ABB RobotStudio station: Solution_1.rspag

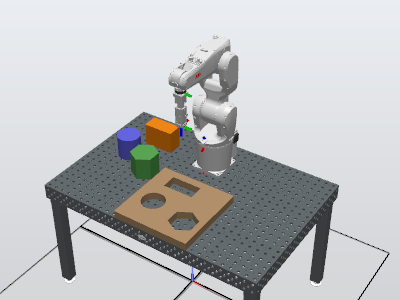
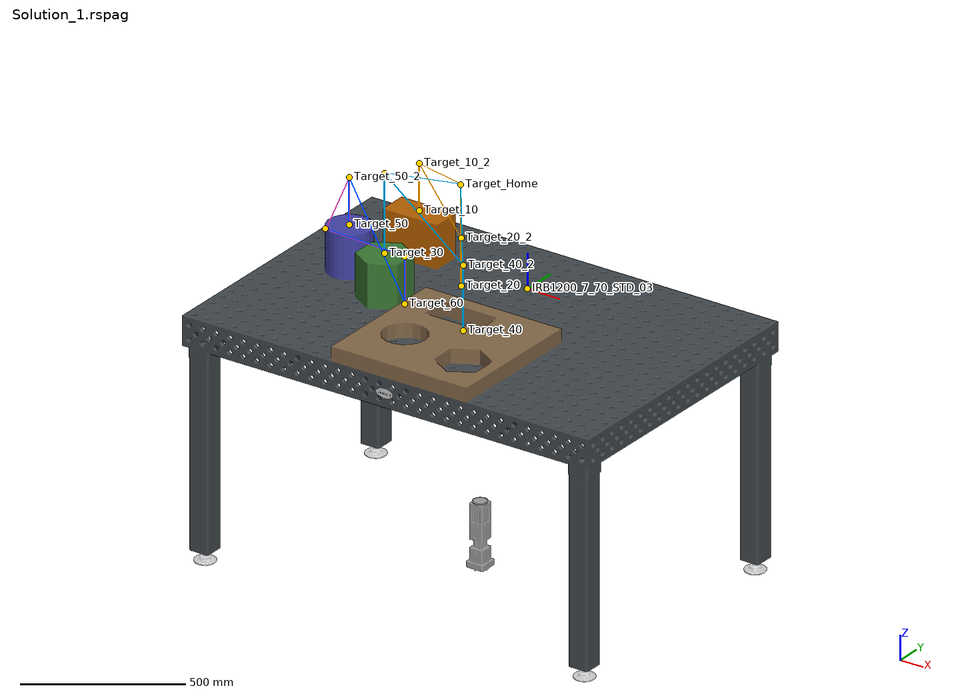
[picture v1: parts stored in the station drawn from their meshes, with robot base, taught points and paths (robot models come from the ABB library and are not in the file)]
--- station ---
Station Solution_1_Tutorial (saved by RobotStudio 22.3.10190.2)
Controller Controller_Solution_1, task T_ROB1: task frame (RAPID world) sits at (0, 250, 830) mm, rotated rx 0 ry 0 rz -90 deg in the station
Controller Controller_Solution_1
  mechanical unit ROB_1: IRB1200_7_70_STD_03, 6 joints, base frame (0, 0, 0) mm
Layout (positions relative to the parent item):
  - table [part] at (-200, -500, 830) mm, size 500 x 500 x 50 mm
  - object_1 [part] at (-600, -150, 830) mm, size 200 x 100 x 150 mm
  - object_2 [part] at (-650, -150, 830) mm, size 149.5 x 149.7 x 150 mm
  - object_3 [part] at (-700, -200, 830) mm, size 155.5 x 179.5 x 150 mm
  - siegmund_1500_1000 [part], size 1500 x 1010.3 x 830 mm
  - object_11 [part] at (-200, -500, 830) mm, size 200 x 100 x 150 mm
  - object_22 [part] at (-200, -500, 830) mm, size 149.5 x 149.7 x 150 mm
  - object_33 [part] at (-200, -500, 830) mm, size 155.5 x 179.5 x 150 mm
  - Assembly2_3 [graphiccomponentgroup] at (-38.87, -9.32, 138.6) mm, rotated rx -90 ry 0 rz 0 deg
    - MHM-32D1-X6400(0):3 [graphiccomponentgroup] at (38.87, 1.1, -15.68) mm, rotated rx 0 ry -90 rz 0 deg
      - _MHM-A3201-1-X6400_DAMPER [part] at (25, -74.2, 0) mm, size 49.7 x 6 x 50 mm
      - _MHM-32D1-X6400(0)_BODY:2 [part] at (25, 0, 25) mm, rotated rx 0 ry 90 rz 0 deg, size 50 x 79.6 x 50 mm
    - M4x10:5 [part] at (39.02, 86.1, -10.68) mm, rotated rx 180 ry 0 rz 0 deg, size 7 x 7 x 14 mm
    - M4x10:7 [part] at (39.02, 36.1, -10.68) mm, rotated rx 180 ry 0 rz 0 deg, size 7 x 7 x 14 mm
    - ITEM30x30x100:3 [part] at (38.87, 106.1, 9.32) mm, rotated rx 0 ry 0 rz -90 deg, size 100 x 30 x 30 mm
    - M5x75:2 [part] at (57.87, 13.1, -9.68) mm, rotated rx -90 ry 0 rz 0 deg, size 8.5 x 8.5 x 25 mm
    - M4x10:8 [part] at (39.02, 86.1, 29.32) mm, size 7 x 7 x 14 mm
    - M4x10:9 [part] at (39.02, 36.1, 29.32) mm, size 7 x 7 x 14 mm
    - M5x75:3 [part] at (19.87, 13.1, 28.32) mm, rotated rx -90 ry 0 rz 0 deg, size 8.5 x 8.5 x 25 mm
    - M5x75:4 [part] at (57.87, 13.1, 28.32) mm, rotated rx -90 ry 0 rz 0 deg, size 8.5 x 8.5 x 25 mm
    - M5x75:5 [part] at (19.87, 13.1, -9.68) mm, rotated rx -90 ry 0 rz 0 deg, size 8.5 x 8.5 x 25 mm
    - KQ2L06-01N:3 [part] at (47.37, -5.7, 30.32) mm, rotated rx 90 ry 0 rz 89.92 deg, size 21.3 x 22.5 x 10.4 mm
    - KQ2L06-01N:4 [part] at (30.37, -64.9, 30.32) mm, rotated rx 90 ry 0 rz 89.92 deg, size 21.3 x 22.5 x 10.4 mm
    - Part_Bottom_Blue:1 [part] at (17.33, 6.1, -15.68) mm, rotated rx 90 ry 0 rz 0 deg, size 50 x 50 x 45 mm
    - Part_Middle_Black:2 [part] at (17.33, 116.1, 34.32) mm, rotated rx -90 ry 0 rz 0 deg, size 50 x 50 x 45 mm
    - Part_Top_Blue:4 [part] at (38.87, 128.6, 9.32) mm, rotated rx 90 ry 0 rz 0 deg, size 63.8 x 63.8 x 17.5 mm
    - M4x25:1 [part] at (19.87, 109.1, -9.68) mm, rotated rx 90 ry 0 rz 0 deg, size 7 x 7 x 29 mm
    - M4x25:2 [part] at (57.87, 109.1, 28.32) mm, rotated rx 90 ry 0 rz 0 deg, size 7 x 7 x 29 mm
    - M4x25:3 [part] at (19.87, 109.1, 28.32) mm, rotated rx 90 ry 0 rz 0 deg, size 7 x 7 x 29 mm
    - M4x25:4 [part] at (57.87, 109.1, -9.68) mm, rotated rx 90 ry 0 rz 0 deg, size 7 x 7 x 29 mm
    - M4_nut:1 [part] at (57.87, 129.7, 28.32) mm, rotated rx 0 ry -14.91 rz 0 deg, size 7 x 2.2 x 8.1 mm
    - M5x16:1 [part] at (50, 128.6, 20.46) mm, rotated rx 90 ry 0 rz 0 deg, size 8.5 x 8.5 x 21 mm
    - M6x16:1 [part] at (63.87, 129.6, 9.32) mm, rotated rx 90 ry 0 rz 0 deg, size 10 x 10 x 22 mm
    - M4_nut:2 [part] at (57.87, 129.7, -9.68) mm, rotated rx 0 ry -14.91 rz 0 deg, size 7 x 2.2 x 8.1 mm
    - M4_nut:3 [part] at (19.87, 129.7, -9.68) mm, rotated rx 0 ry -14.91 rz 0 deg, size 7 x 2.2 x 8.1 mm
    - M4_nut:4 [part] at (19.87, 129.7, 28.32) mm, rotated rx 0 ry -14.91 rz 0 deg, size 7 x 2.2 x 8.1 mm
    - M5x16:2 [part] at (50, 128.6, -1.82) mm, rotated rx 90 ry 0 rz 0 deg, size 8.5 x 8.5 x 21 mm
    - M5x16:3 [part] at (27.73, 128.6, 20.46) mm, rotated rx 90 ry 0 rz 0 deg, size 8.5 x 8.5 x 21 mm
    - M5x16:4 [part] at (27.73, 128.6, -1.82) mm, rotated rx 90 ry 0 rz 0 deg, size 8.5 x 8.5 x 21 mm
    - M6x16:2 [part] at (13.87, 129.6, 9.32) mm, rotated rx 90 ry 0 rz 0 deg, size 10 x 10 x 22 mm
    - M6x16:3 [part] at (38.87, 129.6, -15.68) mm, rotated rx 90 ry 0 rz 0 deg, size 10 x 10 x 22 mm
    - M6x16:4 [part] at (38.87, 129.6, 34.32) mm, rotated rx 90 ry 0 rz 0 deg, size 10 x 10 x 22 mm
  - smc_magnetic_gripper [mechanism] at (0, -101, 1539.1) mm, rotated rx 180 ry 0 rz 90 deg
      TCP smc_magnetic_gripper at (38.87, -79.1, 9.32) mm, rotated rx 90 ry 0 rz 0 deg
      links: Assembly2_3_Merged
  - IRB1200_7_70_STD_03 [mechanism, from %ABB.RobotStudio.Models.IRB1200%\IRB1200_7_70_STD_03.rslib] at (0, 250, 830) mm, rotated rx 0 ry 0 rz -90 deg; joint values [0, 0, 0, 0, 1.5708, 0] (rad or m)
  - Positioner_object_1 [smart component, from Components\Positioner.rslib]
      properties: Object=object_1; Position=[-0.6 -0.15 0.83]; Orientation=[0 0 0]; Reference=Global; ReferenceObject=(none)
  - Attacher_object_1 [smart component, from Components\Attacher.rslib]
      properties: Parent=smc_magnetic_gripper; Flange=0; Child=object_1; Mount=false; Offset=[0 0 0]; Orientation=[0 0 0]
  - Detacher_object_1 [smart component, from Components\Detacher.rslib]
      properties: Child=object_1; KeepPosition=true
  - Positioner_object_2 [smart component, from Components\Positioner.rslib]
      properties: Object=object_2; Position=[-0.65 -0.15 0.83]; Orientation=[0 0 0]; Reference=Global; ReferenceObject=(none)
  - Positioner_object_3 [smart component, from Components\Positioner.rslib]
      properties: Object=object_3; Position=[-0.7 -0.2 0.83]; Orientation=[0 0 0]; Reference=Global; ReferenceObject=(none)
  - Attacher_object_2 [smart component, from Components\Attacher.rslib]
      properties: Parent=smc_magnetic_gripper; Flange=0; Child=object_2; Mount=false; Offset=[0 0 0]; Orientation=[0 0 0]
  - Attacher_object_3 [smart component, from Components\Attacher.rslib]
      properties: Parent=smc_magnetic_gripper; Flange=0; Child=object_3; Mount=false; Offset=[0 0 0]; Orientation=[0 0 0]
  - Detacher_object_2 [smart component, from Components\Detacher.rslib]
      properties: Child=object_2; KeepPosition=true
  - Detacher_object_3 [smart component, from Components\Detacher.rslib]
      properties: Child=object_3; KeepPosition=true
  - Frame_1 [frame] at (0, 0, 217.7) mm
Attachment: smc_magnetic_gripper is attached to IRB1200_7_70_STD_03 / Link6
Station signals: DI reset
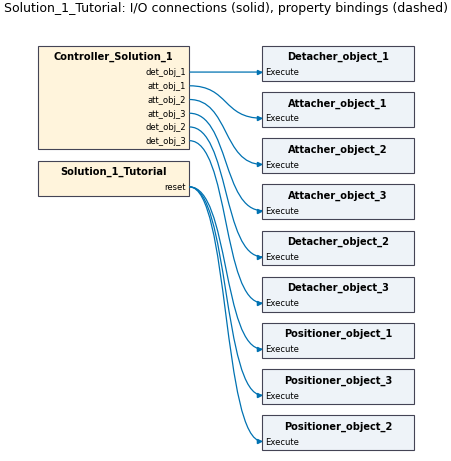
Station logic (signal -> signal, property => property):
  Controller_Solution_1.det_obj_1 -> Detacher_object_1.Execute
  Solution_1_Tutorial.reset -> Positioner_object_1.Execute
  Solution_1_Tutorial.reset -> Positioner_object_3.Execute
  Solution_1_Tutorial.reset -> Positioner_object_2.Execute
  Controller_Solution_1.att_obj_1 -> Attacher_object_1.Execute
  Controller_Solution_1.att_obj_2 -> Attacher_object_2.Execute
  Controller_Solution_1.att_obj_3 -> Attacher_object_3.Execute
  Controller_Solution_1.det_obj_2 -> Detacher_object_2.Execute
  Controller_Solution_1.det_obj_3 -> Detacher_object_3.Execute
Targets, tools, work objects and paths stored in the station and not in the controller backup, written as RAPID:
! task T_ROB1
MODULE CalibData
  PERS tooldata MyTool:=[TRUE,[[31.792631019,0,229.638935148],[0.945518576,0,0.325568154,0]],[1,[0,0,1],[1,0,0,0],0,0,0]];
ENDMODULE


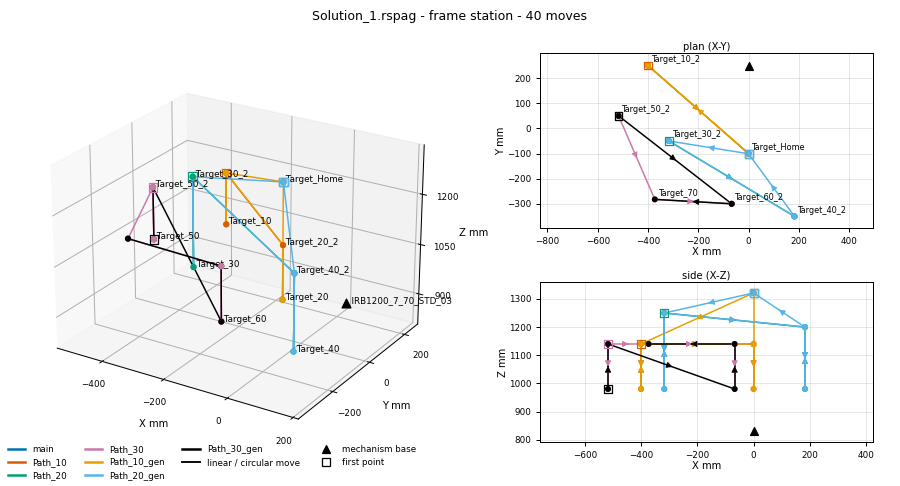
[picture p0: tool path of Solution_1.rspag in frame station, 40 of 40 moves have a stored position in this frame; points joined in program order, loops and branches not executed]
--- Backups/Controller_Solution_1/RAPID/TASK1/PROGMOD/CalibData.modx ---
MODULE CalibData
    PERS tooldata smc_magnetic_gripper:=[TRUE,[[0,0,217.7],[1,0,0,0]],[0.72,[0.001,0.267,107.779],[1,0,0,0],0,0,0]];
ENDMODULE

--- Backups/Controller_Solution_1/RAPID/TASK1/PROGMOD/Module1.modx ---
MODULE Module1
        CONST robtarget Target_Home:=[[351,0,491.4],[0,0,1,0],[-1,0,-1,0],[9E+09,9E+09,9E+09,9E+09,9E+09,9E+09]];
    CONST robtarget Target_10_2:=[[0,-400,310],[0,0,1,0],[-1,0,-2,0],[9E+09,9E+09,9E+09,9E+09,9E+09,9E+09]];
    CONST robtarget Target_10:=[[0,-400,150],[0,0,1,0],[-1,0,-2,0],[9E+09,9E+09,9E+09,9E+09,9E+09,9E+09]];
    CONST robtarget Target_20_2:=[[350,0,310],[0,0,1,0],[0,0,0,0],[9E+09,9E+09,9E+09,9E+09,9E+09,9E+09]];
    CONST robtarget Target_20:=[[350,0,150],[0,0,1,0],[0,0,-1,0],[9E+09,9E+09,9E+09,9E+09,9E+09,9E+09]];
    CONST robtarget Target_30_2:=[[300,-317.298,420],[0,0,1,0],[0,0,0,0],[9E+09,9E+09,9E+09,9E+09,9E+09,9E+09]];
    CONST robtarget Target_30:=[[300,-317.298,150],[0,0,1,0],[0,0,0,0],[9E+09,9E+09,9E+09,9E+09,9E+09,9E+09]];
    CONST robtarget Target_40_2:=[[600,182.702,370],[0,0,1,0],[0,0,0,0],[9E+09,9E+09,9E+09,9E+09,9E+09,9E+09]];
    CONST robtarget Target_40:=[[600,182.702,150],[0,0,1,0],[0,0,0,0],[9E+09,9E+09,9E+09,9E+09,9E+09,9E+09]];
    CONST robtarget Target_50_2:=[[200,-517.298,310],[0,0,1,0],[0,0,0,0],[9E+09,9E+09,9E+09,9E+09,9E+09,9E+09]];
    CONST robtarget Target_60:=[[550,-67.298,150],[0,0,1,0],[0,0,0,0],[9E+09,9E+09,9E+09,9E+09,9E+09,9E+09]];
    CONST robtarget Target_60_2:=[[550,-67.298,310],[0,0,1,0],[0,0,0,0],[9E+09,9E+09,9E+09,9E+09,9E+09,9E+09]];
    CONST robtarget Target_70:=[[532.420048745,-372.921595913,310],[0,0,1,0],[0,0,0,0],[9E+09,9E+09,9E+09,9E+09,9E+09,9E+09]];
    CONST robtarget Target_50:=[[200,-517.298,150],[0,0,1,0],[-1,0,-1,0],[9E+09,9E+09,9E+09,9E+09,9E+09,9E+09]];

!***********************************************************
    !
    ! Module:  Module1
    !
    ! Description:
    !   <Insert description here>
    !
    ! Author: gruna
    !
    ! Version: 1.0
    !
    !***********************************************************


    !***********************************************************
    !
    ! Procedure main
    !
    !   This is the entry point of your program
    !
    !***********************************************************
    PROC main()
        !MoveL Target_Home,v500,z100,smc_magnetic_gripper\WObj:=wobj0;
        MoveL Target_Home,v300,z100,smc_magnetic_gripper\WObj:=wobj0;
        Path_10;
        Path_20;
        Path_30;
        MoveL Target_Home,v300,z100,smc_magnetic_gripper\WObj:=wobj0;
    ENDPROC
    PROC Path_10()
        MoveL Target_10_2,v500,z100,smc_magnetic_gripper\WObj:=wobj0;
        MoveL Target_10,v500,fine,smc_magnetic_gripper\WObj:=wobj0;
        PulseDO att_obj_1;
        WaitTime 0.5;
        MoveL Target_10_2,v500,z100,smc_magnetic_gripper\WObj:=wobj0;
        MoveL Target_20_2,v500,z20,smc_magnetic_gripper\WObj:=wobj0;
        MoveL Target_20,v500,fine,smc_magnetic_gripper\WObj:=wobj0;
        PulseDO det_obj_1;
        WaitTime 0.5;
    ENDPROC
    PROC Path_20()
        MoveL Target_30_2,v400,z100,smc_magnetic_gripper\WObj:=wobj0;
        MoveL Target_30,v400,fine,smc_magnetic_gripper\WObj:=wobj0;
        PulseDO att_obj_3;
        WaitTime 0.5;
        MoveL Target_30_2,v400,z50,smc_magnetic_gripper\WObj:=wobj0;
        MoveL Target_40_2,v400,z20,smc_magnetic_gripper\WObj:=wobj0;
        MoveL Target_40,v400,fine,smc_magnetic_gripper\WObj:=wobj0;
        PulseDO det_obj_3;
        WaitTime 0.5;
        MoveL Target_40_2,v400,z100,smc_magnetic_gripper\WObj:=wobj0;
    ENDPROC
    PROC Path_30()
        MoveL Target_50_2,v400,z100,smc_magnetic_gripper\WObj:=wobj0;
        MoveL Target_50,v400,fine,smc_magnetic_gripper\WObj:=wobj0;
        PulseDO att_obj_2;
        WaitTime 0.5;
        MoveL Target_50_2,v400,z100,smc_magnetic_gripper\WObj:=wobj0;
        MoveL Target_70,v400,z100,smc_magnetic_gripper\WObj:=wobj0;
        MoveL Target_60_2,v400,z20,smc_magnetic_gripper\WObj:=wobj0;
        MoveL Target_60,v400,fine,smc_magnetic_gripper\WObj:=wobj0;
        PulseDO det_obj_2;
        WaitTime 0.5;
        MoveL Target_60_2,v400,z100,smc_magnetic_gripper\WObj:=wobj0;
    ENDPROC

    PROC Path_10_gen()
        MoveL Target_Home,v500,z100,smc_magnetic_gripper\WObj:=wobj0;
        MoveL Target_10_2,v500,z100,smc_magnetic_gripper\WObj:=wobj0;
        MoveL Target_10,v500,fine,smc_magnetic_gripper\WObj:=wobj0;
        PulseDO att_obj_1;
        WaitTime 1;
        MoveL Target_10_2,v500,z100,smc_magnetic_gripper\WObj:=wobj0;
        MoveL Target_20_2,v500,z100,smc_magnetic_gripper\WObj:=wobj0;
        MoveL Target_20,v500,fine,smc_magnetic_gripper\WObj:=wobj0;
        PulseDO det_obj_1;
        WaitTime 1;
        MoveL Target_Home,v500,z100,smc_magnetic_gripper\WObj:=wobj0;
    ENDPROC
    PROC Path_20_gen()
        MoveL Target_Home,v400,z100,smc_magnetic_gripper\WObj:=wobj0;
        MoveL Target_30_2,v400,z100,smc_magnetic_gripper\WObj:=wobj0;
        MoveL Target_30,v400,fine,smc_magnetic_gripper\WObj:=wobj0;
        MoveL Target_30_2,v400,z100,smc_magnetic_gripper\WObj:=wobj0;
        MoveL Target_40_2,v400,z100,smc_magnetic_gripper\WObj:=wobj0;
        MoveL Target_40,v400,fine,smc_magnetic_gripper\WObj:=wobj0;
        MoveL Target_40_2,v400,z100,smc_magnetic_gripper\WObj:=wobj0;
        MoveL Target_Home,v400,z100,smc_magnetic_gripper\WObj:=wobj0;
    ENDPROC
    PROC Path_30_gen()
        MoveL Target_50,v1000,z100,smc_magnetic_gripper\WObj:=wobj0;
        MoveL Target_50_2,v1000,z100,smc_magnetic_gripper\WObj:=wobj0;
        MoveL Target_60,v1000,z100,smc_magnetic_gripper\WObj:=wobj0;
        MoveL Target_60_2,v1000,z100,smc_magnetic_gripper\WObj:=wobj0;
        MoveL Target_70,v1000,z100,smc_magnetic_gripper\WObj:=wobj0;
    ENDPROC
ENDMODULE

--- Backups/Controller_Solution_1/SYSPAR/EIO.cfg ---
EIO:CFG_1.0:7:0::
#
EIO_SIGNAL:

      -Name "att_obj_1" -SignalType "DO"

      -Name "det_obj_1" -SignalType "DO"

      -Name "att_obj_2" -SignalType "DO"

      -Name "att_obj_3" -SignalType "DO"

      -Name "det_obj_2" -SignalType "DO"

      -Name "det_obj_3" -SignalType "DO"

#CTRL_SIGNATURE:PSStGgkjFbik+b14gifOdyMVyZFRnqFFprYa3ZiZExG8xUJI4yYsM99kzr8D5kZDYVoFTbCg+iEJyTPvN/r9lw==

--- Backups/Controller_Solution_1/SYSPAR/PROC.cfg ---
PROC:CFG_1.0:7:0::

#CTRL_SIGNATURE:I+y2QaV15gWtHGM+5Z4idi3NiusZu29hLyokxM3ohwogLM8MfydOTWOtI2G6szFitByh5svEYsXD7agPogo+dQ==
